ABB RobotStudio station: Autoclasiffier_Vacuostato_20181219-100423.rsstn

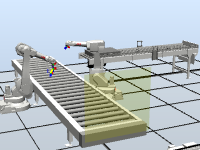
Station Station (saved by RobotStudio 6.6.7701.1025)
Controller Sistema12, task T_ROB1: task frame (RAPID world) sits at (920, -1100, 0) mm, rotated rx 0 ry 0 rz 180 deg in the station
Controller Sistema10, task T_ROB1: task frame (RAPID world) sits at (-920, -900, 0) mm in the station
Controller Sistema10
  mechanical unit ROB_1: JUAN, 6 joints, base frame (0, 0, 0) mm
Controller Sistema12
  mechanical unit ROB_1: ROBERTO, 6 joints, base frame (0, 0, 0) mm
Layout (positions relative to the parent item):
  - JUAN [mechanism, from Robots\IRB1600_6_145_G_02.rslib] at (-920, -900, 0) mm; joint values [-0.0666, 0.1032, 0.3482, 0, 1.1194, 3.075] (rad or m)
  - ROBERTO [mechanism, from Robots\IRB1600_6_145_G_02.rslib] at (920, -1100, 0) mm, rotated rx 0 ry 0 rz 180 deg; joint values [-0.4677, 0.0079, -0.0561, 0.0825, 1.1142, -0.2191] (rad or m)
  - 600_guide [part, from Equipment\Conveyor Guide 600.rslib] at (3800, 50, 0) mm, rotated rx 0 ry 0 rz 180 deg
  - 4800_3str_h2 [part, from Equipment\Conveyor 4800 3str h2.rslib] at (0, -5364.61, 0) mm
  - 950_4800_h2 [part, from Equipment\Conveyor 950 4800 h2.rslib] at (475, -3400, 0) mm, rotated rx 0 ry 0 rz 90 deg
  - Pieza_5 [part] at (920, -500, 775) mm
  - Componente inteligente_1 [smart component]
      signals: DI dedo_Juan, DO Aspira
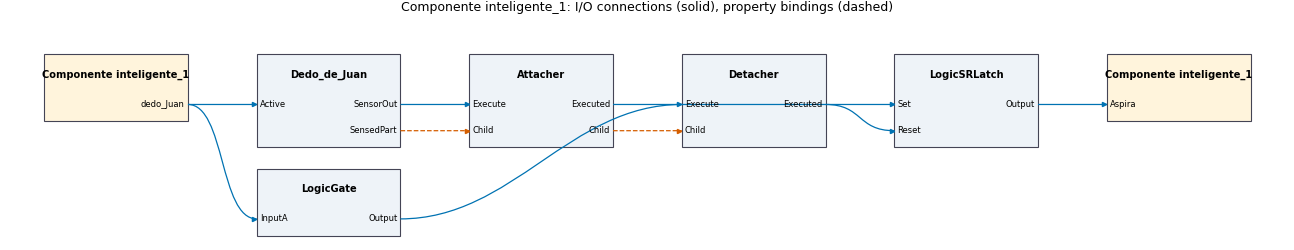
      connections:
        Dedo_de_Juan.SensorOut -> Attacher.Execute
        LogicGate.Output -> Detacher.Execute
        Componente inteligente_1.dedo_Juan -> Dedo_de_Juan.Active
        Componente inteligente_1.dedo_Juan -> LogicGate.InputA
        Attacher.Executed -> LogicSRLatch.Set
        LogicSRLatch.Output -> Componente inteligente_1.Aspira
        Detacher.Executed -> LogicSRLatch.Reset
        Dedo_de_Juan.SensedPart => Attacher.Child
        Attacher.Child => Detacher.Child
    - Dedo_de_Roberto [smart component, from Components\LineSensor.rslib] at (0, 0, 0) mm
        properties: Start=[0 0 0]; End=[0 0 0.035]; Radius=0.002; SensedPart=(none); SensedPoint=[0.215981719970703 -0.749844604492187 1.15866088867188]
      - _sensorPart_ [part]
    - Attacher [smart component, from Components\Attacher.rslib]
        properties: Parent=(none); Flange=0; Child=Pieza_7; Mount=false; Offset=[0 0 0]; Orientation=[0 0 0]
    - LogicGate [smart component, from Components\LogicGate.rslib] at (-1050.67, 0, 0) mm
        properties: Operator=NOT; Delay=0
    - Dedo_de_Juan [smart component, from Components\LineSensor.rslib] at (-159.7, -950.69, 856.04) mm, rotated rx -180 ry 0 rz 0 deg
        properties: Start=[0 0 0.08]; End=[0 0 0.11]; Radius=0.002; SensedPart=Pieza_7; SensedPoint=[-0.209697967529297 -0.95068701171875 0.706042236328125]
      - _sensorPart_ [part]
    - Detacher [smart component, from Components\Detacher.rslib]
        properties: Child=Pieza_7; KeepPosition=true
    - LogicSRLatch [smart component, from Components\LogicSRLatch.rslib]
  - chasis_t [part] at (-230, -1000, 595) mm, rotated rx 180 ry 0 rz 90 deg
  - Pieza_6 [part] at (370, -1250, 415) mm, rotated rx 0 ry -90 rz 0 deg
  - Componente inteligente_2 [smart component]
  - T_Chasis [part] at (0, 0, 100) mm
  - Componente inteligente_3 [smart component]
      signals: DI Montaje_acabado, DO Sensor, DI on
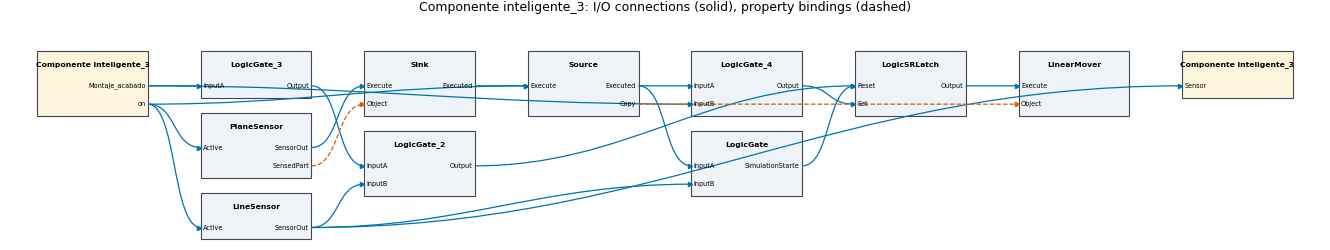
      connections:
        PlaneSensor.SensorOut -> Sink.Execute
        LogicSRLatch.Output -> LinearMover.Execute
        Source.Executed -> LogicGate.InputA
        LineSensor.SensorOut -> LogicGate.InputB
        Componente inteligente_3.Montaje_acabado -> LogicGate_3.InputA
        LogicGate_3.Output -> LogicGate_2.InputA
        LineSensor.SensorOut -> LogicGate_2.InputB
        LogicGate_2.Output -> LogicSRLatch.Reset
        Source.Executed -> LogicGate_4.InputA
        Componente inteligente_3.Montaje_acabado -> LogicGate_4.InputB
        LogicGate_4.Output -> LogicSRLatch.Set
        LineSensor.SensorOut -> Componente inteligente_3.Sensor
        Sink.Executed -> Source.Execute
        Componente inteligente_3.on -> Source.Execute
        SimulationEvents.SimulationStarted -> LogicSRLatch.Reset
        Componente inteligente_3.on -> PlaneSensor.Active
        Componente inteligente_3.on -> LineSensor.Active
        PlaneSensor.SensedPart => Sink.Object
        Source.Copy => LinearMover.Object
    - Source [smart component, from Components\Source.rslib]
        properties: Source=T_Chasis; Copy=(none); Parent=(none); Position=[0 2.5 0]; Orientation=[0 0 0]; Transient=false; PhysicsBehavior=0
    - PlaneSensor [smart component, from Components\PlaneSensor.rslib]
        properties: Origin=[-0.52 -3.6 0.35]; Axis1=[0 0 1]; Axis2=[1.05 0 0]; SensedPart=(none)
      - _sensorPart_ [part]
    - Sink [smart component, from Components\Sink.rslib]
        properties: Object=(none)
    - LinearMover [smart component, from Components\LinearMover.rslib]
        properties: Object=(none); Direction=[0 -0.001 0]; Speed=0.5; Reference=Global; ReferenceObject=(none)
    - LineSensor [smart component, from Components\LineSensor.rslib]
        properties: Start=[0.040738 -1.264377 0.404542]; End=[0.040738 -1.264377 0.42054]; Radius=0.001; SensedPart=(none); SensedPoint=[0 0 0]
      - _sensorPart_ [part]
    - LogicSRLatch [smart component, from Components\LogicSRLatch.rslib]
    - LogicGate_2 [smart component, from Components\LogicGate.rslib]
        properties: Operator=AND; Delay=0
    - LogicGate_3 [smart component, from Components\LogicGate.rslib]
        properties: Operator=NOT; Delay=0
    - LogicGate_4 [smart component, from Components\LogicGate.rslib]
        properties: Operator=OR; Delay=0
  - Mano_de_Juan [mechanism] at (-159.7, -950.69, 856.04) mm, rotated rx -180 ry 0 rz 0 deg
      TCP Mano_de_Juan at (0, 0, 100) mm
      links: Pieza_7
Attachment: Mano_de_Juan is attached to JUAN / Link6
Attachment: Dedo_de_Juan is attached to Mano_de_Juan / Pieza_7
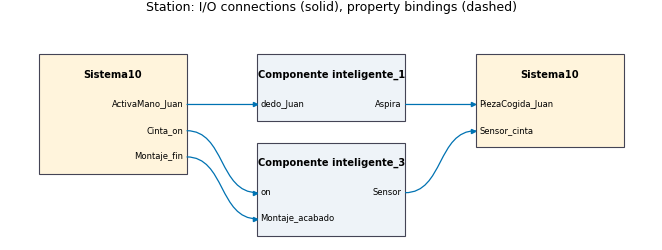
Station logic (signal -> signal, property => property):
  Componente inteligente_1.Aspira -> Sistema10.PiezaCogida_Juan
  Sistema10.ActivaMano_Juan -> Componente inteligente_1.dedo_Juan
  Sistema10.Cinta_on -> Componente inteligente_3.on
  Componente inteligente_3.Sensor -> Sistema10.Sensor_cinta
  Sistema10.Montaje_fin -> Componente inteligente_3.Montaje_acabado
Targets, tools, work objects and paths stored in the station, written as RAPID:
! task T_ROB1
MODULE Module1
  CONST robtarget Target_10:=[[710.302,-50.687,666.042],[0,1,0,0],[-1,0,1,0],[9E+09,9E+09,9E+09,9E+09,9E+09,9E+09]];
  CONST robtarget Target_20:=[[760.301980587,-50.686989693,756.042035513],[-0.000000033,1,-0.000000027,0.000000018],[-1,-1,1,0],[9E+09,9E+09,9E+09,9E+09,9E+09,9E+09]];
  PROC Path_10()
    MoveL Target_10,v1000,z100,Mano_de_Juan\WObj:=wobj0;
    SetDO ActivaMano_Juan,1;
    MoveL Target_20,v1000,z100,Mano_de_Juan\WObj:=wobj0;
  ENDPROC
ENDMODULE

! task T_ROB1
MODULE CalibData
  PERS tooldata Mano_de_Juan:=[TRUE,[[0,0,100],[1,0,0,0]],[1,[0,0,1],[1,0,0,0],0,0,0]];
ENDMODULE

